(* CoDeSys 2.3 export: VARIAVEIS_RESTRITAS.EXP *)

(* Global variable list: variaveis_restritas *)
VAR_GLOBAL CONSTANT
	CREDIT_STRING_ROW: ARRAY [1..4] OF STRING := 'DESENVOLVIDO POR:', 'NATANAEL JOSUE RABELLO', 'TECNICO ELETRONICO PROGRAMADOR', 'EMAIL:NATANAELX10@HOTMAIL.COM';
	CREDIT_SIZE: ARRAY [1..4] OF USINT := 17, 22, 30, 29; (*numero de caracteres das strings acima*)
END_VAR
(* NAO APAGUE AQUI - RESTRITO*)
